FUNCTION_BLOCK Test_NotificationHandlerOnlyAddedOnce EXTENDS T_UnitTestBase
VAR
    Notification        : T_Notification;
    NotificationHandler : T_NotificationHandler;
    IsRaised            : BOOL;
END_VAR

METHOD  Init
VAR_INPUT
END_VAR
END_METHOD

{attribute 'analysis' := '-33'} // inhibit unused variable warning
METHOD RunTest
NotificationHandler.FB_init(bInitRetains := FALSE,
                            bInCopyCode  := FALSE);

Notification
    .ClearNotificationHandlers()
    .AddNotificationHandler(NotificationHandler)
    .AddNotificationHandler(NotificationHandler);

Notification.Raise();
IsRaised := NotificationHandler.IsRaised();

AssertIsTrue(Condition := IsRaised = TRUE,
             Message   := 'IsRaised is not true');

IsRaised := NotificationHandler.IsRaised();

AssertIsTrue(Condition := IsRaised = FALSE,
             Message   := 'IsRaised is not false');

TestCompleted := TRUE;
END_METHOD

END_FUNCTION_BLOCK

(* stored: Version 1.1.0.1, ProductVersion 3.1.4024.12
   POU Test_NotificationHandlerOnlyAddedOnce: Id {d822493b-b417-457e-b68d-ce48b3adc9d5}, SpecialFunc None
   Method Init: Id {4682e57e-171d-4766-990e-46f6a03e0e82}
   Method RunTest: Id {e4801cbe-a69b-4c40-b3f3-077fc4956321} *)
